Staubli VAL3: avaAdvMoveIndex.pgx

program avaAdvMoveIndex(num& x_nIndex)
  local num l_nIndex
begin

  //return the first available "advanced move" index...-1 if max moves reached
  for l_nIndex=0 to size(bAdvMoveBusy)-1
    if !bAdvMoveBusy[l_nIndex]
      x_nIndex=l_nIndex
      return
    endIf
  endFor
  x_nIndex=-1

end
